// TIA Portal V17 export
// export: Created 2024-09-02T12:50:34.6849322Z, ExportSetting WithDefaults, DisplayName Totally Integrated Automation Portal, DisplayVersion V17, DisplayName TIA Portal Openness, DisplayVersion V17, DisplayName TIA Portal Version Control Interface, DisplayVersion V17, DisplayName STEP 7 Professional, DisplayVersion V17, DisplayName STEP 7 Safety, DisplayVersion V17, DisplayName WinCC Professional, DisplayVersion V17
TYPE "typ_Anbauteil"
// stored: IsFailsafeCompliant false
   STRUCT
      BauteilTyp : Array[1..11] of Char;   // Typskennzeichnung / Type designation
      ErstesZeichen : Byte;   // Nummer des ersten Zeichens zur Auswertung / Number of the first character for evaluation
      Laenge : Byte;   // Laenge aller Zeichen zur Auswertung / Length of all characters for evaluation
   END_STRUCT;
END_TYPE
